FUNCTION_BLOCK INTERNAL FINAL FB_WriteBytesTests EXTENDS FB_TestSuite
VAR_INPUT
END_VAR
VAR_OUTPUT
END_VAR
VAR
END_VAR

ShouldWriteBytesTheory();

METHOD PRIVATE ShouldWriteBytes
VAR_IN_OUT CONSTANT    
    aExpectedBytes  : ARRAY[0..31] OF BYTE;
    aBytesToWrite   : ARRAY[*] OF BYTE;
END_VAR
VAR_INPUT CONSTANT
    nBufferPosStart     : UDINT;
    nExpectedBufferPos  : UDINT;
END_VAR
VAR_INST
    fbCtx   : FB_WriteContext;
END_VAR
VAR
    aActualBytes : ARRAY[0..31] OF BYTE;
    hrActual : HRESULT; 
    nLength : UDINT;
END_VAR

// Arrange
fbCtx.FromBuffer(aActualBytes);
fbCtx.refCtx.stState.nBufferPos := nBufferPosStart;
nLength := TO_UDINT(UPPER_BOUND(aBytesToWrite, 1) + 1);

// Act
{warning disable C0041}
hrActual := F_WriteBytes(fbCtx.refCtx, aBytesToWrite, nLength);

// Assert
AssertEquals_DINT(
     Expected:= S_OK,
     Actual:= hrActual,
     Message:= 'Expected S_OK instead of error');

AssertArrayEquals_BYTE(
    Expecteds:= aExpectedBytes,
    Actuals:= aActualBytes,
    Message:= '');
    
AssertEquals_UDINT(
    Expected:= nExpectedBufferPos,
    Actual:= fbCtx.refCtx.stState.nBufferPos,
    Message:= CONCAT('Expected stState.nBufferPos to equal ', TO_STRING(nExpectedBufferPos)));
END_METHOD

METHOD PRIVATE ShouldWriteBytesTheory
VAR CONSTANT
    cExpectedBytesTest1     : ARRAY[0..31] OF BYTE := [16#00, 16#03, 16#01, 16#02, 16#03];
    cBytesToWriteTest1      : ARRAY[0..2] OF BYTE := [16#01, 16#02, 16#03];
END_VAR
TEST(__POUNAME());

ShouldWriteBytes(aExpectedBytes:= cExpectedBytesTest1, aBytesToWrite:= cBytesToWriteTest1, nBufferPosStart:= 1, nExpectedBufferPos:= 5);

TEST_FINISHED_NAMED(__POUNAME());
END_METHOD

END_FUNCTION_BLOCK

(* stored: Version 1.1.0.1
   POU FB_WriteBytesTests: Id {623a6450-385e-49a5-8d3f-af9fc8d6603b}, SpecialFunc None
   Method ShouldWriteBytes: Id {6c4f2652-46fa-445e-9fae-34e5a74bdcfe}
   Method ShouldWriteBytesTheory: Id {6aa9646c-8353-4e06-a43c-4b32755f577b} *)
